INTERFACE ITF_Regelschuif_In_DG

METHOD get : SINT
VAR_INPUT
END_VAR
END_METHOD

END_INTERFACE

(* stored: Version 1.1.0.1, ProductVersion 3.1.4026.8
   Itf ITF_Regelschuif_In_DG: Id {a1595fe7-c7ae-46d5-a51e-360ac0f615ce}
   Method get: Id {164dc5d0-07cc-482b-ba0a-5a29f959989f} *)
